(* PLC project pusher, Dassault Systèmes ControlBuild 2024x *)
(* stored: creationDateTime 2023-10-04T11:03:51-01:00 *)

FUNCTION_BLOCK motion_lib.pusher
  VAR_INPUT
    moveX : REAL := 0.0;
    moveY : REAL := 0.0;
    moveZ : REAL := 0.0;
  END_VAR
  VAR
    status_act_prod : DINT := 0;
    m11 : REAL := 1.0;
    m12 : REAL := 0.0;
    m13 : REAL := 0.0;
    m14 : REAL := 0.0;
    m21 : REAL := 0.0;
    m22 : REAL := 1.0;
    m23 : REAL := 0.0;
    m24 : REAL := 0.0;
    m31 : REAL := 0.0;
    m32 : REAL := 0.0;
    m33 : REAL := 1.0;
    m34 : REAL := 0.0;
    m41 : REAL := 0.0;
    m42 : REAL := 0.0;
    m43 : REAL := 0.0;
    m44 : REAL := 1.0;
    moveX1 : REAL := 0.0;
    moveY1 : REAL := 0.0;
    moveZ1 : REAL := 0.0;
  END_VAR
  VAR CONSTANT
    oriX : REAL := 1.0;
    oriY : REAL := 1.0;
    oriZ : REAL := 1.0;
  END_VAR

moveX1 := moveX * oriX ;
moveY1 := moveY * oriY;
moveZ1 := moveZ * oriZ ;
moveBy(myself, moveX1 ,moveY1 , moveZ1);
END_FUNCTION_BLOCK
